FUNCTION_BLOCK PUBLIC FB_Socket
VAR_OUTPUT
	bActive		: BOOL;
END_VAR

PROPERTY PUBLIC Active : BOOL
GET
Active := bActive;
END_GET
END_PROPERTY

METHOD PUBLIC Off
bActive := false;
END_METHOD

METHOD PUBLIC On
bActive := true;
END_METHOD

END_FUNCTION_BLOCK

(* stored: Version 1.1.0.1, ProductVersion 3.1.4024.12
   POU FB_Socket: Id {bcd0fc7b-8f02-4944-8c70-a0fd855e493d}, SpecialFunc None
   Property Active: Id {7b6f0e6d-2dbd-47ae-93da-62a9512b93b9}
   Get Get: Id {8c8b66f5-16dc-4037-91bb-575e9eb6568e}
   Method Off: Id {c7ff13f2-11a8-49a5-b53c-943873250584}
   Method On: Id {82ac724e-ad77-4a02-9fbd-75e46d868f7e} *)
